FUNCTION_BLOCK PresenceSensor IMPLEMENTS ITF_BinarySensor
VAR_INPUT
END_VAR
VAR_OUTPUT
END_VAR
VAR
	DI_WPDetected AT %I* : BOOL;
END_VAR

PROPERTY Value : BOOL
GET
Value := DI_WPDetected;
END_GET
END_PROPERTY

END_FUNCTION_BLOCK

(* stored: Version 1.1.0.1, ProductVersion 3.1.4024.4
   POU PresenceSensor: Id {198d39e5-5ee9-4fa6-a367-84fcc42193f6}, SpecialFunc None
   Property Value: Id {03f98580-06f3-40ed-ac76-171736b50910}
   Get Get: Id {8365c618-6d09-4a92-a9c3-fd6075546b66} *)
